FUNCTION TryConvert_LWORD_TO_DWORD : BOOL
VAR_INPUT
	in : LWORD;
	out : REFERENCE TO DWORD;
END_VAR

IF in > DatatypeLimits.MAX_VALUE_OF_LWORD_WHICH_CAN_BE_HELD_IN_A_DWORD THEN
	RETURN;
END_IF

out := LWORD_TO_DWORD(in);
TryConvert_LWORD_TO_DWORD := TRUE;

END_FUNCTION

(* stored: Version 1.1.0.1, ProductVersion 3.1.4024.12
   POU TryConvert_LWORD_TO_DWORD: Id {179b288d-c10c-41af-b68a-fd3f8f36a01d}, SpecialFunc None *)
